// TIA Portal V17 export
// export: Created 2025-03-10T13:11:42.9078584Z, ExportSetting WithDefaults, DisplayName Totally Integrated Automation Portal, DisplayVersion V17 Update 8, DisplayName TIA Portal Openness, DisplayVersion V17 Update 8, DisplayName TIA Portal Version Control Interface, DisplayVersion V17, DisplayName SINAMICS Startdrive Advanced, DisplayVersion V17 SP2, DisplayName SINAMICS Startdrive G110M, G120, G120C, G120D, G120P, G115D, DisplayVersion V17 SP2, DisplayName SINAMICS Startdrive G130, G150, S120, S150, SINAMICS MV, S210, DisplayVersion V17 SP2, DisplayName STEP 7 Professional, DisplayVersion V17 Update 8, DisplayName SINUMERIK ONE STEP 7 Toolbox, DisplayVersion V17 Update 12, DisplayName SINUMERIK 840D sl STEP 7 Toolbox, DisplayVersion V17 Update 12, DisplayName STEP 7 Safety, DisplayVersion V17 Update 6, DisplayName WinCC Advanced, DisplayVersion V17 Update 8
DATA_BLOCK "DB7215_PART_TYPE"   // DB7215
{ S7_Optimized_Access := 'FALSE'; DB_Accessible_From_OPC_UA := 'FALSE' }
AUTHOR : ETXETAR
VERSION : 1.0
// stored: AutoNumber false, DBAccessibleFromOPCUA false, DBAccessibleFromWebserver true, IsOnlyStoredInLoadMemory false, IsWriteProtectedInAS false
   VAR RETAIN
      GENERAL_CONDITIONS : Bool;   // GENERAL CONDITIONS
      AUTO_PART_TYPE : Bool;   // AUTO PART TYPE SELECT
      REQUEST_NEW_PART_TYPE : Bool;   // REQUEST NEW PART TYPE
      COMMAND : Bool;   // COMMAND
      REQUEST_HELP : Bool;   // REQUEST HELP
      SPARE : Byte;
      PART_TYPE_01_SELECTED : Bool;   // PART TYPE 1 SELECTED
      PART_TYPE_02_SELECTED : Bool;   // PART TYPE 2 SELECTED
      PART_TYPE_03_SELECTED : Bool;   // PART TYPE 3 SELECTED
      PART_TYPE_04_SELECTED : Bool;   // PART TYPE 4 SELECTED
      PART_TYPE_05_SELECTED : Bool;   // PART TYPE 5 SELECTED
      PART_TYPE_06_SELECTED : Bool;   // PART TYPE 6 SELECTED
      PART_TYPE_07_SELECTED : Bool;   // PART TYPE 7 SELECTED
      PART_TYPE_08_SELECTED : Bool;   // PART TYPE 8 SELECTED
      PART_TYPE_09_SELECTED : Bool;   // PART TYPE 9 SELECTED
      PART_TYPE_10_SELECTED : Bool;   // PART TYPE 10 SELECTED
      PART_TYPE_11_SELECTED : Bool;   // PART TYPE 11 SELECTED
      PART_TYPE_12_SELECTED : Bool;   // PART TYPE 12 SELECTED
      PART_TYPE_13_SELECTED : Bool;   // PART TYPE 13 SELECTED
      PART_TYPE_14_SELECTED : Bool;   // PART TYPE 14 SELECTED
      PART_TYPE_15_SELECTED : Bool;   // PART TYPE 15 SELECTED
      PART_TYPE_16_SELECTED : Bool;   // PART TYPE 16 SELECTED
      PART_TYPE_17_SELECTED : Bool;   // PART TYPE 17 SELECTED
      PART_TYPE_18_SELECTED : Bool;   // PART TYPE 18 SELECTED
      PART_TYPE_19_SELECTED : Bool;   // PART TYPE 19 SELECTED
      PART_TYPE_20_SELECTED : Bool;   // PART TYPE 20 SELECTED
      PART_TYPE_21_SELECTED : Bool;   // PART TYPE 21 SELECTED
      PART_TYPE_22_SELECTED : Bool;   // PART TYPE 22 SELECTED
      PART_TYPE_23_SELECTED : Bool;   // PART TYPE 23 SELECTED
      PART_TYPE_24_SELECTED : Bool;   // PART TYPE 24 SELECTED
      PART_TYPE_25_SELECTED : Bool;   // PART TYPE 25 SELECTED
      PART_TYPE_26_SELECTED : Bool;   // PART TYPE 26 SELECTED
      PART_TYPE_27_SELECTED : Bool;   // PART TYPE 27 SELECTED
      PART_TYPE_28_SELECTED : Bool;   // PART TYPE 28 SELECTED
      PART_TYPE_29_SELECTED : Bool;   // PART TYPE 29 SELECTED
      PART_TYPE_30_SELECTED : Bool;   // PART TYPE 30 SELECTED
      PART_TYPE_31_SELECTED : Bool;   // PART TYPE 31 SELECTED
      PART_TYPE_32_SELECTED : Bool;   // PART TYPE 32 SELECTED
      PART_TYPE_SEL_FAULT : Bool;   // PART TYPE SELECTED GANTRY FAULT / PART TYPE SELECTED FAULT
      NO_PART_TYPE_SELECTED : Bool;   // NO PART TYPE SELECTED
      PART_TYPE_U01_FIXTURES : Bool;   // PART TYPE FIXTURE 1 / PART TYPE UNIT 01 FIXTURES
      PART_TYPE_U02_FIXTURES : Bool;   // PART TYPE FIXTURE 2 / PART TYPE UNIT 02 FIXTURES
      PART_TYPE_U03_FIXTURES : Bool;   // PART TYPE MEASURE UNIT FIXTURES
      PART_TYPE_F4 : Bool;   // PART TYPE FIXTURE 4
      PART_TYPE_F5 : Bool;   // PART TYPE FIXTURE 5
      PART_TYPE_ONE_PART : Bool;   // PART TYPE ONE LONG PART
      PART_TYPE_TWO_PARTS : Bool;   // PART TYPE TWO SHORT PARTS
      IS : Bool;   // IMMEDIATE STOP ALARMS
      IS_SEOC : Bool;   // IMMEDIATE STOP & STOP AT END OF CYCLE ALARMS
      RHP : Bool;   // RETURN TO HOME POSITION ALARMS
      RHP_SEOC : Bool;   // RETURN TO HOME POSITION & STOP AT END OF CYCLE ALARMS
      SEOC : Bool;   // STOP AT END OF CYCLE ALARMS
      IS_WARNING : Bool;   // IMMEDIATE STOP WARNING
      RHP_WARNING : Bool;   // RETURN TO HOME POSITION WARNING
      SEOC_WARNING : Bool;   // STOP AT END OF CYCLE WARNING
      WARNING : Bool;   // WARNING
      HELP : Bool;   // HELP
      PART_TYPE_SEQ_WARNING : Bool;   // PART TYPE SEQ WARNING
      REQUEST_CHANGE_TYPE : Bool;   // REQUEST CHANGE TYPE
      MECH_ACKNOW_REQUIRED : Bool;   // MECH ACKNOW REQUIRED
      PART_TYPE_SCREEN : Bool;   // PART TYPE SCRREN SELECTED / PART TYPE SCREEN SELECTED
      ANY_PART_TYPE_FAULT : Bool;   // ANY PART TYPE FAULT
      ANY_PART_TYPE_OK : Bool;   // ANY PART TYPE OK
      DISCORDANCY_P_TYPE_1 : Bool;   // DISCORDANCY PART TYPE1 AND PARTS
      DISCORDANCY_P_TYPE_2 : Bool;   // DISCORDANCY PART TYPE2 AND PARTS
      DISCORDANCY_P_TYPE_3 : Bool;   // DISCORDANCY PART TYPE3 AND PARTS
      CONDITIONS_HELP : Bool;   // CONDITIONS HELP
      PART_TYPE : Int;
      Part_Type_Low : Byte;   // PART TYPE LOW
      Part_Type_High : Byte;   // PART TYPE HIGH
      Mach_Part_Type_Selected : Int;   // MACHINE PART TYPE SELECTED
      Gantry_Part_Loaded : Int;   // GANTRY PART LOADED
      TIMER_PART_SELECTION : TON_TIME;   // PART SELECTION ALARM TIMER
   END_VAR
BEGIN
   TIMER_PART_SELECTION.PT := T#500ms;
END_DATA_BLOCK
